// TwinCAT 3 PLC project PLC
// ProgramVersion: 3.1.4023.0
// libraries:
//   Tc2_Standard, * (Beckhoff Automation GmbH)
//   Tc2_System, * (Beckhoff Automation GmbH)
//   Tc2_Utilities, * (Beckhoff Automation GmbH)
//   Tc3_Module, * (Beckhoff Automation GmbH)
// project tree:
//   / PlcTask.TcTTO
//   POUs/ MAIN.TcPOU
// real-time tasks:
//   TASK PlcTask: cycle T#10ms, priority 20, ADS port 350
// I/O:
//   DEVICE Device 2 (USB) (disabled)
//     Box 0 (CPX8XX)
//   DEVICE Device 1 (EtherCAT) (disabled), AmsNetId 172.16.17.1.2.1
//     Term 1 (EK1814) [EK1814 EtherCAT IO-Coupler  (1A E-Bus, 4 Ch. Dig. In, 3ms, 4 Ch. Dig. Out 24V, 0,5A)]
// variable links:
//   PLC Instance <-> Device 1 (EtherCAT)/Term 1 (EK1814)
//     PlcTask Inputs/MAIN.DigitalInputForPB1 <-> Channel 1/Input
//   PLC Instance <-> Device 2 (USB)/Box 0 (CPX8XX)
//     PlcTask Inputs/MAIN.USBInputForPB1 <-> Term 2 (CPx9xx-8)/Channel 1/Key 1

CONFIGURATION PLC
    RESOURCE PLC ON TwinCAT3
        TASK PlcTask(INTERVAL := T#10ms, PRIORITY := 20);
        PROGRAM MAIN WITH PlcTask : MAIN;
    END_RESOURCE
END_CONFIGURATION

// ---- POUs/MAIN.TcPOU
PROGRAM MAIN
VAR
	DigitalInputForPB1	AT%I*	:BOOL;

	USBInputForPB1		AT%I*	:BOOL;

	PushButton1					:BOOL;
	Counter						:DINT;
	
	xRestartTwinCAT				:BOOL;
	fbResetTwinCAT				:TC_Restart;
END_VAR
VAR CONSTANT
	{IF defined (EC_PB)}
		sActiveVariant				:STRING:='EC_PB';
	{ELSIF defined (USB_PB)}
		sActiveVariant				:STRING:='USB_PB';
	{END_IF}	
END_VAR

{IF defined (EC_PB)}
	PushButton1:=DigitalInputForPB1;
	Counter:=Counter+1;
{ELSIF defined (USB_PB)}
	PushButton1:=USBInputForPB1;
	Counter:=Counter-1;
{END_IF}

fbResetTwinCAT(
	NETID:='' , 
	RESTART:=xRestartTwinCAT);

END_PROGRAM
